FUNCTION_BLOCK FB_SolSpringPiston_2Pos
(* Single-solenoid, spring-return 2-position actuator.
   Coil energised  -> drives to EXTENDED.
   Coil de-energised -> mechanical spring returns to RETRACTED.

   The coil is a continuous force against the spring, so Section 2 uses a
   LATCH-and-RETAIN pattern: the coil is set TRUE on Extend command and
   FALSE on Retract command, and RETAINS its state (via VAR_OUTPUT retain)
   any cycle no explicit command is active. Without the latch the coil
   would drop the moment the extended sensor fires and the spring would
   immediately pull the piston back.

   Fail-safe by construction: broken wire, dead coil, PLC power loss
   or e-stop all leave bOutSolenoid FALSE and the spring retracts.

   Interface is kept symmetric with FB_SolSolPiston_2Pos so a sequencer FB
   (e.g. FB_PistonAutoCycle) can drive either actuator type without a
   custom variant. Reuses ST_HmiPiston unchanged; the retract-coil mirror
   field (stHmi.bOutSolenoidRetract) is always FALSE because no retract
   coil exists on this actuator. *)
VAR_INPUT
    (* Automatic Commands from PLC sequence logic. Wired to FALSE in MAIN until FB_Auto exists. *)
    bAutoCmdExtend    : BOOL;
    bAutoCmdRetract   : BOOL;

    (* External jog request (e.g. panel push-button). OR-merged with the
       HMI's stHmi.bManJogExtend inside so a physical PB and the HMI
       button can drive the same jog without stepping on each other.
       Only takes effect while eMode = Manual (same gate as the HMI jog). *)
    bJogExtend        : BOOL;

    (* Physical Feedback (Proximity Switches) *)
    bSwitchExtended   : BOOL;
    bSwitchRetracted  : BOOL;
END_VAR

VAR_IN_OUT
    (* HMI contract — mode, manual + simulate inputs, latched + sensor status *)
    stHmi             : ST_HmiPiston;
END_VAR

VAR_OUTPUT
    (* Physical Output to Solenoid — SINGLE coil.
       TRUE  = coil energised, actuator drives EXTENDED.
       FALSE = coil de-energised, spring returns actuator to RETRACTED. *)
    bOutSolenoid      : BOOL;
END_VAR

VAR
    (* Internal Target States *)
    bTargetExtend     : BOOL;
    bTargetRetract    : BOOL;

    (* HMI Manual-Button Edge Detection *)
    fbTrigManExtend   : R_TRIG;
    fbTrigManRetract  : R_TRIG;

    (* Effective sensor states = real OR HMI simulate. Recomputed every cycle in Section 0a. *)
    bSwitchExtended_eff  : BOOL;
    bSwitchRetracted_eff : BOOL;

    (* Previous-cycle snapshots for the mode-field bridge in Section 0b.
       Classic PLC HMI writes stHmi.bMode (Rotary Switch is boolean-only);
       web HMI writes stHmi.eMode (enum via ToggleSwitch). This FB is the
       authoritative reader of eMode, so we sync in whichever direction
       changed since last cycle. *)
    bPrevMode : BOOL;
    ePrevMode : E_ControlMode;
END_VAR

(* ==========================================
   0b. MODE-FIELD BRIDGE — sync bMode <-> eMode
   The classic PLC HMI (VISUs) writes stHmi.bMode because its Rotary Switch
   element is boolean-only. FlowerPyHmi writes stHmi.eMode over ADS.
   (The retired Flower_HMI web project did the same via a ToggleSwitch.) Rest of this FB reads eMode as the authoritative field,
   so we mirror bMode into eMode when the classic HMI toggled the switch,
   and mirror eMode back into bMode when the web HMI (or anyone else) wrote
   eMode. Edge-triggered — whichever side changed since last cycle wins.
   Runs BEFORE Section 0 so downstream logic sees a coherent eMode.
   ========================================== *)
IF stHmi.bMode <> bPrevMode THEN
    // Classic VISU changed bMode → propagate to eMode
    IF stHmi.bMode THEN
        stHmi.eMode := E_ControlMode.Automatic;
    ELSE
        stHmi.eMode := E_ControlMode.Manual;
    END_IF;
ELSIF stHmi.eMode <> ePrevMode THEN
    // Web HMI (or any other writer) changed eMode → propagate to bMode
    stHmi.bMode := (stHmi.eMode = E_ControlMode.Automatic);
END_IF;

bPrevMode := stHmi.bMode;
ePrevMode := stHmi.eMode;

(* ==========================================
   0a. EFFECTIVE SENSOR INPUTS (real OR HMI simulate)
   ========================================== *)
bSwitchExtended_eff  := bSwitchExtended  OR stHmi.bSimulateExtended;
bSwitchRetracted_eff := bSwitchRetracted OR stHmi.bSimulateRetracted;

(* ==========================================
   0. HMI MANUAL BUTTON LATCHING (Radio-Button Behavior)
   ========================================== *)
fbTrigManExtend(CLK := stHmi.bManCmdExtend);
fbTrigManRetract(CLK := stHmi.bManCmdRetract);

// Independent IFs (not ELSIF): if multiple edges fire in the same cycle, the last one wins (Retract > Extend).
IF fbTrigManExtend.Q  THEN stHmi.bSelectedExtend := TRUE;  stHmi.bSelectedRetract := FALSE; END_IF;
IF fbTrigManRetract.Q THEN stHmi.bSelectedExtend := FALSE; stHmi.bSelectedRetract := TRUE;  END_IF;

IF stHmi.eMode = E_ControlMode.Automatic THEN
    stHmi.bSelectedExtend := FALSE; stHmi.bSelectedRetract := FALSE;
END_IF;

(* ==========================================
   1. MODE SELECTION & COMMAND MAPPING
   Spring-return semantics: both bAutoCmd* inputs are accepted for interface
   parity with FB_SolSolPiston_2Pos, but physically only Extend commands the
   coil. If both auto bits are TRUE we treat it as a conflict and de-energise
   (safe default — spring retracts).
   ========================================== *)
IF stHmi.eMode = E_ControlMode.Automatic THEN
    bTargetExtend  := bAutoCmdExtend  AND NOT bAutoCmdRetract;
    bTargetRetract := bAutoCmdRetract AND NOT bAutoCmdExtend;

ELSIF stHmi.eMode = E_ControlMode.Manual THEN
    bTargetExtend  := stHmi.bSelectedExtend;
    bTargetRetract := stHmi.bSelectedRetract;

ELSE
    // Safe default: undefined mode → no targets
    bTargetExtend  := FALSE;
    bTargetRetract := FALSE;
END_IF;

(* ==========================================
   1a. JOG OVERRIDE — clear latched selection while either jog is held
   ========================================== *)
// Section 1 above already copied stHmi.bSelected* into bTarget*. The stale
// bTarget* is harmless because Section 2's jog branches sit ahead of the
// bTarget* branches in the IF/ELSIF ladder and preempt them.
IF stHmi.bManJogExtend OR stHmi.bManJogRetract OR bJogExtend THEN
    stHmi.bSelectedExtend := FALSE; stHmi.bSelectedRetract := FALSE;
END_IF;

(* ==========================================
   1b. TARGET-REACHED RESET — clear bSelected* once the piston arrives
   ========================================== *)
IF stHmi.bSelectedExtend  AND bSwitchExtended_eff  THEN stHmi.bSelectedExtend  := FALSE; END_IF;
IF stHmi.bSelectedRetract AND bSwitchRetracted_eff THEN stHmi.bSelectedRetract := FALSE; END_IF;

(* ==========================================
   2. SOLENOID CONTROL — single coil, LATCH-and-RETAIN
   The coil is a continuous force against the spring. If it drops, the spring
   wins and the actuator retracts. So the coil must be LATCHED TRUE from the
   moment Extend is commanded until Retract is commanded — not pulsed until
   the sensor fires (which is the double-solenoid pattern).
   Structure:
     - Jog branches first, gated by Manual mode.
     - Explicit Extend / Retract command branches drive the coil to a
       definite state.
     - The IF ladder has NO ELSE. When no branch matches, VAR_OUTPUT retain
       semantics carry the coil forward:
         * At the Extended sensor after a successful extend (Section 1b just
           cleared bTargetExtend) → coil retains TRUE → piston HOLDS.
         * At the Retracted sensor after a successful retract → coil retains
           FALSE → piston HOLDS retracted (spring already there).
         * Sequencer DWELL_EXT (both auto bits FALSE) → coil retains TRUE
           for the full dwell instead of releasing the piston.
     - No sensor guards on the drive branches: holding the coil TRUE while
       at the Extended sensor is normal operation, not a wasted drive.
   Fail-safe still holds: cold boot, PLC reset, or e-stop leave bOutSolenoid
   at its default FALSE and the spring retracts.
   ========================================== *)
// JOG EXTEND: while held in Manual, energise coil. HMI-owned bManJogExtend
// OR external bJogExtend (panel push-button) -- both share the Manual gate.
IF (stHmi.bManJogExtend OR bJogExtend) AND stHmi.eMode = E_ControlMode.Manual THEN
    bOutSolenoid := TRUE;

// JOG RETRACT: while held in Manual, de-energise coil (spring retracts)
ELSIF stHmi.bManJogRetract AND stHmi.eMode = E_ControlMode.Manual THEN
    bOutSolenoid := FALSE;

// EXTEND commanded — energise coil (latched via retain when bTargetExtend clears)
ELSIF bTargetExtend THEN
    bOutSolenoid := TRUE;

// RETRACT commanded — de-energise coil, spring retracts
ELSIF bTargetRetract THEN
    bOutSolenoid := FALSE;

// No branch → bOutSolenoid RETAINS its previous value (see block header).
END_IF;

(* ==========================================
   3. HMI STATUS FEEDBACK
   bIsMoving is derived from sensor state alone: with Section 2's latch
   semantics, bOutSolenoid stays TRUE at the extended limit — so ORing
   it in would report "moving" while the piston is actually parked.
   "Between the two limits" is accurate for both strokes: coil-driven
   extend and spring-driven retract both traverse that gap.

   bOutSolenoidRetract is written FALSE unconditionally — no retract coil
   exists on a spring-return actuator, so the mirror stays cleared.
   ========================================== *)
stHmi.bIsExtended         := bSwitchExtended_eff;
stHmi.bIsRetracted        := bSwitchRetracted_eff;
stHmi.bIsMoving           := NOT bSwitchExtended_eff AND NOT bSwitchRetracted_eff;
stHmi.bOutSolenoidExtend  := bOutSolenoid;
stHmi.bOutSolenoidRetract := FALSE;

END_FUNCTION_BLOCK

(* stored: Version 1.1.0.1, ProductVersion 3.1.4026.18
   POU FB_SolSpringPiston_2Pos: Id {dbca3142-cfb0-4b0e-af16-d67fa4f955fc}, SpecialFunc None *)
